// TIA Portal V18 export
TYPE "PLCtoMES_SubCheckIn"
// stored: IsFailsafeCompliant false
   STRUCT
      "P-SubPartID" : String[48];   // 子零件ID，用于和主工件实物ID或虚拟ID绑定,上一个子零件ID绑定完成后需要清空后再写入下一个子零件ID，不能采取覆盖的方式
      "P-SubPartReq" : Bool;   // PLC请求绑定子关重零件验证绑定标志位（关重件SN序列号刷新后触发），MES置位M-SubPartOK或M-SubPartNG信号后，由PLC复位此信号。
      Reserve : Array[1..247] of Byte;   // SubPartReq子零件绑定交互预留
   END_STRUCT;
END_TYPE
